(* Logix 5000 project; controller Corte_Silla vendor 1 type 14 code 156 rev 30.11; software revision 30.00 *)

TASK MainTask (continuous, watchdog 500 ms) : MainProgram

MODULES
   Local : vendor 1 type 14 code 156 (Compact 0, rev 30.11)
END_MODULES

PROGRAM MainProgram   (* main routine Memorizacion_de_etapas *)
VAR
   A1 : BOOL;   // Banda 1
   A2 : BOOL;   // Banda 2
   A3 : BOOL;   // Gripper
   Cont1 : COUNTER := (PRE := 36);
   Cont2 : COUNTER := (PRE := 36);
   Cont3 : COUNTER := (PRE := 36);
   Cont4 : COUNTER := (PRE := 5);
   Cont5 : COUNTER := (PRE := 2);
   Cont6 : COUNTER;
   DI_01 : BOOL;
   DI_02 : BOOL;
   DI_03 : BOOL;
   DI_04 : BOOL;
   DI_05 : BOOL;
   DI_06 : BOOL;
   DI_07 : BOOL;
   DI_08 : BOOL;
   DI_09 : BOOL;
   DI_10 : BOOL;
   DO_01 : BOOL;
   DO_02 : BOOL;
   DO_03 : BOOL;
   DO_04 : BOOL;
   DO_05 : BOOL;
   DO_06 : BOOL;
   DO_07 : BOOL;
   DO_08 : BOOL;
   DO_09 : BOOL;
   DO_10 : BOOL;
   Dobladora_DN : BOOL;
   E0 : BOOL;
   E1 : BOOL;
   E10 : BOOL;
   E11 : BOOL;
   E12 : BOOL;
   E13 : BOOL;
   E14 : BOOL;
   E15 : BOOL;
   E16 : BOOL;
   E17 : BOOL;
   E18 : BOOL;
   E19 : BOOL;
   E2 : BOOL;
   E20 : BOOL;
   E21 : BOOL;
   E22 : BOOL;
   E23 : BOOL;
   E3 : BOOL;
   E4 : BOOL;
   E5 : BOOL;
   E6 : BOOL;
   E7 : BOOL;
   E8 : BOOL;
   E9 : BOOL;
   March : BOOL;
   S1 : BOOL;   // Sensor Banda
   S2 : BOOL;   // Sensor_Dobladora
   Start : BOOL;
   Stop : BOOL;
   T01 : TIMER := (PRE := 100);
   T02 : TIMER := (PRE := 1000);
   Test1 : BOOL;
   Test2 : BOOL;
   Test3 : BOOL;
END_VAR

ROUTINE Activacion_de_salidas   (* ladder *)
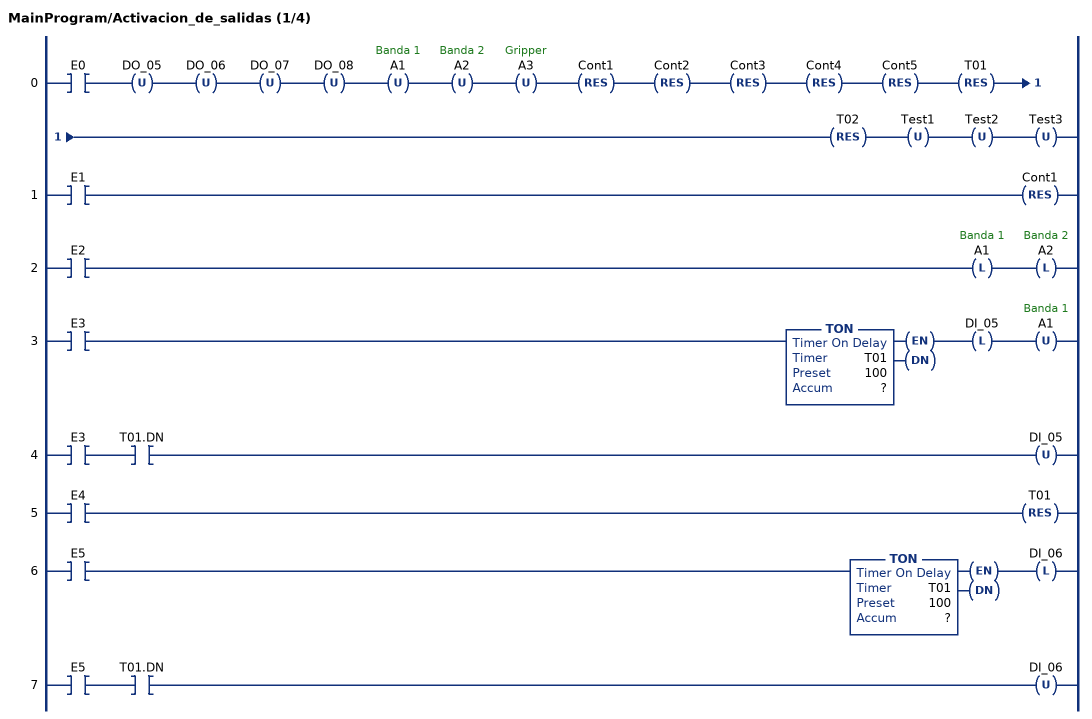
   0: XIC(E0)OTU(DO_05)OTU(DO_06)OTU(DO_07)OTU(DO_08)OTU(A1)OTU(A2)OTU(A3)RES(Cont1)RES(Cont2)RES(Cont3)RES(Cont4)RES(Cont5)RES(T01)RES(T02)OTU(Test1)OTU(Test2)OTU(Test3);
   1: XIC(E1)RES(Cont1);
   2: XIC(E2)OTL(A1)OTL(A2);
   3: XIC(E3)TON(T01,?,?)OTL(DI_05)OTU(A1);
   4: XIC(E3)XIC(T01.DN)OTU(DI_05);
   5: XIC(E4)RES(T01);
   6: XIC(E5)TON(T01,?,?)OTL(DI_06);
   7: XIC(E5)XIC(T01.DN)OTU(DI_06);
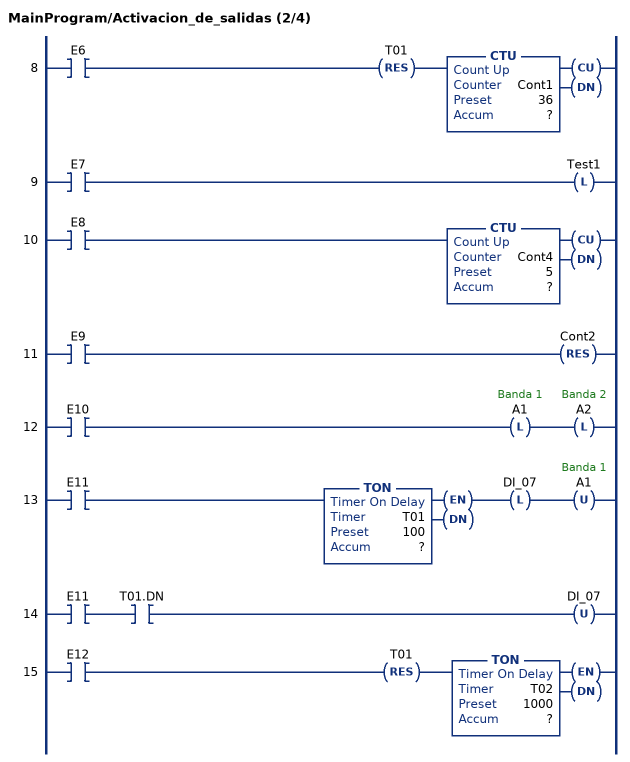
   8: XIC(E6)RES(T01)CTU(Cont1,?,?);
   9: XIC(E7)OTL(Test1);
   10: XIC(E8)CTU(Cont4,?,?);
   11: XIC(E9)RES(Cont2);
   12: XIC(E10)OTL(A1)OTL(A2);
   13: XIC(E11)TON(T01,?,?)OTL(DI_07)OTU(A1);
   14: XIC(E11)XIC(T01.DN)OTU(DI_07);
   15: XIC(E12)RES(T01)TON(T02,?,?);
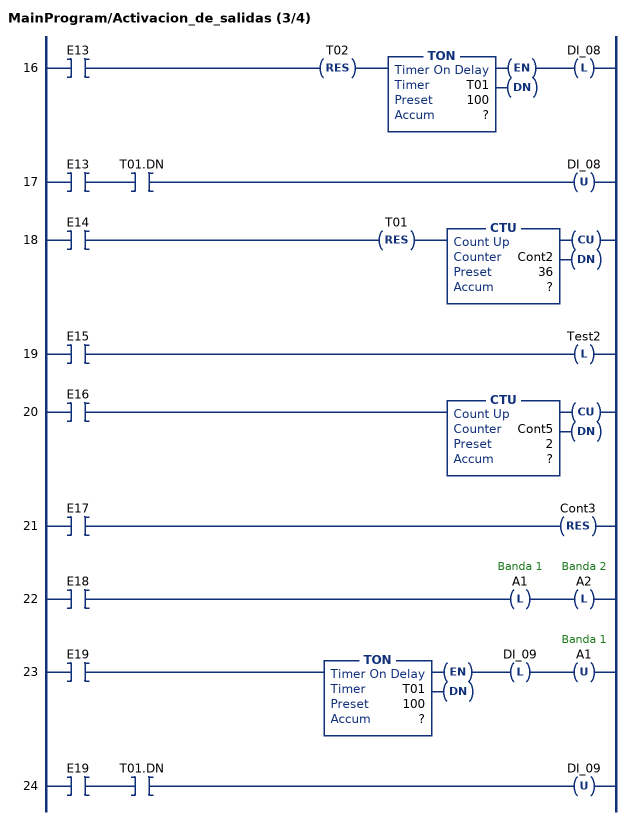
   16: XIC(E13)RES(T02)TON(T01,?,?)OTL(DI_08);
   17: XIC(E13)XIC(T01.DN)OTU(DI_08);
   18: XIC(E14)RES(T01)CTU(Cont2,?,?);
   19: XIC(E15)OTL(Test2);
   20: XIC(E16)CTU(Cont5,?,?);
   21: XIC(E17)RES(Cont3);
   22: XIC(E18)OTL(A1)OTL(A2);
   23: XIC(E19)TON(T01,?,?)OTL(DI_09)OTU(A1);
   24: XIC(E19)XIC(T01.DN)OTU(DI_09);
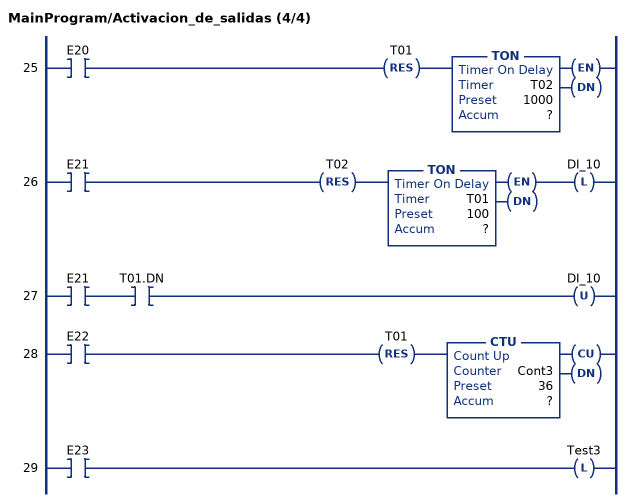
   25: XIC(E20)RES(T01)TON(T02,?,?);
   26: XIC(E21)RES(T02)TON(T01,?,?)OTL(DI_10);
   27: XIC(E21)XIC(T01.DN)OTU(DI_10);
   28: XIC(E22)RES(T01)CTU(Cont3,?,?);
   29: XIC(E23)OTL(Test3);
END_ROUTINE

ROUTINE Memorizacion_de_etapas   (* ladder *)
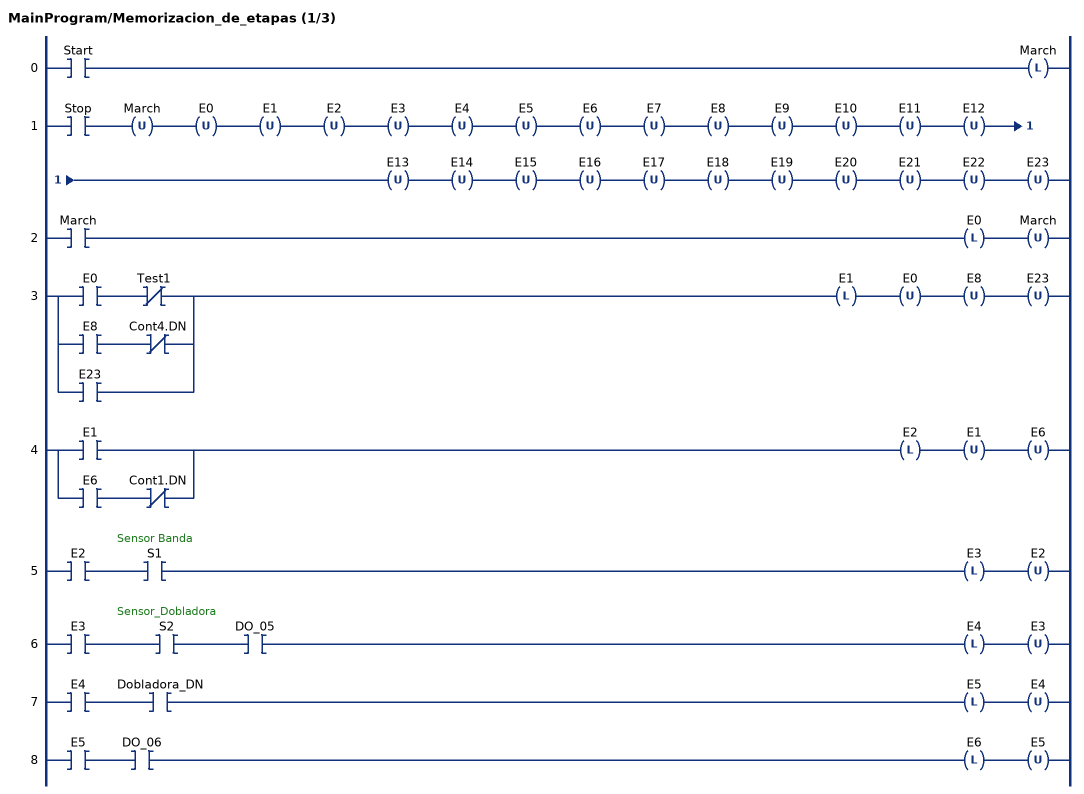
   0: XIC(Start)OTL(March);
   1: XIC(Stop)OTU(March)OTU(E0)OTU(E1)OTU(E2)OTU(E3)OTU(E4)OTU(E5)OTU(E6)OTU(E7)OTU(E8)OTU(E9)OTU(E10)OTU(E11)OTU(E12)OTU(E13)OTU(E14)OTU(E15)OTU(E16)OTU(E17)OTU(E18)OTU(E19)OTU(E20)OTU(E21)OTU(E22)OTU(E23);
   2: XIC(March)OTL(E0)OTU(March);
   3: [XIC(E0) XIO(Test1) ,[XIC(E8) XIO(Cont4.DN) ,XIC(E23) ] ]OTL(E1)OTU(E0)OTU(E8)OTU(E23);
   4: [XIC(E1) ,XIC(E6) XIO(Cont1.DN) ]OTL(E2)OTU(E1)OTU(E6);
   5: XIC(E2)XIC(S1)OTL(E3)OTU(E2);
   6: XIC(E3)XIC(S2)XIC(DO_05)OTL(E4)OTU(E3);
   7: XIC(E4)XIC(Dobladora_DN)OTL(E5)OTU(E4);
   8: XIC(E5)XIC(DO_06)OTL(E6)OTU(E5);
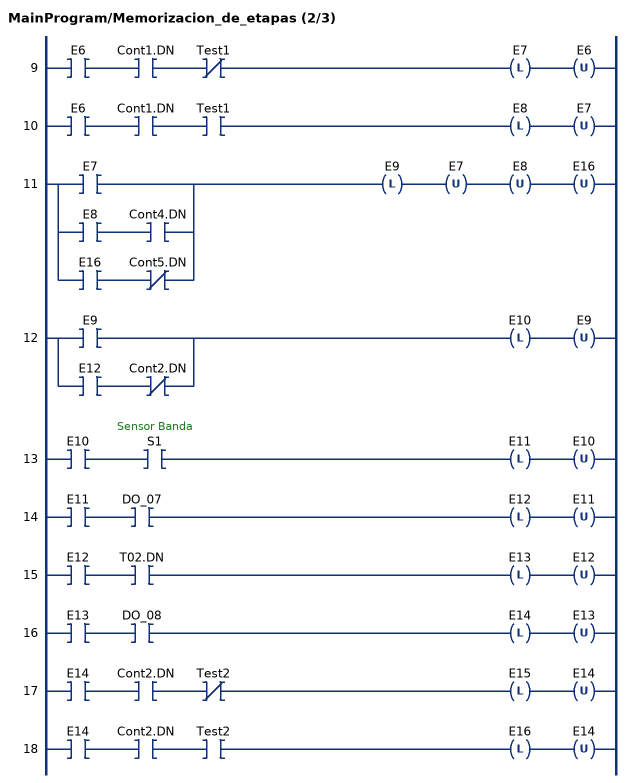
   9: XIC(E6)XIC(Cont1.DN)XIO(Test1)OTL(E7)OTU(E6);
   10: XIC(E6)XIC(Cont1.DN)XIC(Test1)OTL(E8)OTU(E7);
   11: [XIC(E7) ,[XIC(E8) XIC(Cont4.DN) ,XIC(E16) XIO(Cont5.DN) ] ]OTL(E9)OTU(E7)OTU(E8)OTU(E16);
   12: [XIC(E9) ,XIC(E12) XIO(Cont2.DN) ]OTL(E10)OTU(E9);
   13: XIC(E10)XIC(S1)OTL(E11)OTU(E10);
   14: XIC(E11)XIC(DO_07)OTL(E12)OTU(E11);
   15: XIC(E12)XIC(T02.DN)OTL(E13)OTU(E12);
   16: XIC(E13)XIC(DO_08)OTL(E14)OTU(E13);
   17: XIC(E14)XIC(Cont2.DN)XIO(Test2)OTL(E15)OTU(E14);
   18: XIC(E14)XIC(Cont2.DN)XIC(Test2)OTL(E16)OTU(E14);
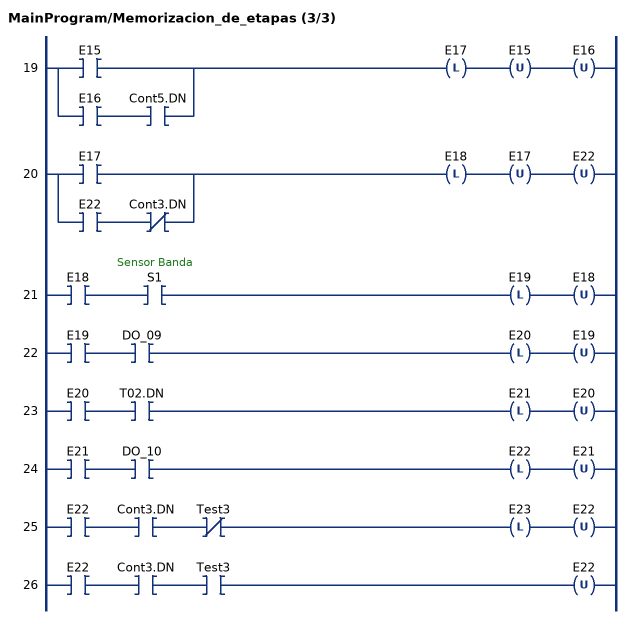
   19: [XIC(E15) ,XIC(E16) XIC(Cont5.DN) ]OTL(E17)OTU(E15)OTU(E16);
   20: [XIC(E17) ,XIC(E22) XIO(Cont3.DN) ]OTL(E18)OTU(E17)OTU(E22);
   21: XIC(E18)XIC(S1)OTL(E19)OTU(E18);
   22: XIC(E19)XIC(DO_09)OTL(E20)OTU(E19);
   23: XIC(E20)XIC(T02.DN)OTL(E21)OTU(E20);
   24: XIC(E21)XIC(DO_10)OTL(E22)OTU(E21);
   25: XIC(E22)XIC(Cont3.DN)XIO(Test3)OTL(E23)OTU(E22);
   26: XIC(E22)XIC(Cont3.DN)XIC(Test3)OTU(E22);
END_ROUTINE
END_PROGRAM
